(* PLC project {project_name}, OpenIXl generator OpenIXL generator v0.1 *)
(* stored: companyURL https://github.com/Bleebop/IXL_project, creationDateTime {creation_date_time}, modificationDateTime {creation_date_time} *)

TYPE TC : (NIL := -1);
END_TYPE

TYPE SWITCH : (NIL := -1);
END_TYPE

TYPE SIGNAL : (NIL := -1);
END_TYPE

TYPE TRAIN_STATE : STRUCT
  exists : BOOL;
  rear_pos : TC;
  front_pos : TC;
  orientation : DIR;
  stopped : BOOL;
END_STRUCT;
END_TYPE

TYPE DIR : (NIL := -1, DOWN := 0, UP := 1);
END_TYPE

TYPE SW_POS_t : (NIL := -1, LEFT := 1, RIGHT := 2, INTERMEDIATE := 3);
END_TYPE

TYPE ENTRY_POINT_t : STRUCT
  tc : TC;
  orientation : DIR;
END_STRUCT;
END_TYPE

TYPE EXIT_POINT_t : STRUCT
  tc : TC;
  orientation : DIR;
END_STRUCT;
END_TYPE

TYPE ROUTE : (NIL := -1);
END_TYPE

PROGRAM safety_PLC
  VAR
    route_state : ARRAY[1..const_g.nRoute] OF route_state;
    Approaching_train : ARRAY[1..const_g.nRoute] OF Approaching_train;
    switch_locked : ARRAY[1..const_g.nSwitch] OF BOOL;
    switch_required_left : ARRAY[1..const_g.nSwitch] OF BOOL;
    switch_required_right : ARRAY[1..const_g.nSwitch] OF BOOL;
  END_VAR
  VAR CONSTANT
    DELAY_DESTRUCT : ARRAY[1..const_g.nRoute] OF TIME := [];
  END_VAR
  VAR_OUTPUT
    route_open : ARRAY[1..const_g.nRoute] OF BOOL;
    route_entry_authorization : ARRAY[1..const_g.nRoute] OF BOOL;  (* The starting signal of the route can be opened to go through this route *)
    signal_open_maneuver : ARRAY[1..const_g.nSignal] OF BOOL;  (* Signal is opened for CBTC trains (downstream block occupation is ignored) *)
    switch_command_left : ARRAY[1..const_g.nSwitch] OF BOOL;
    switch_command_right : ARRAY[1..const_g.nSwitch] OF BOOL;
  END_VAR

(* FBD diagram, written out as Structured Text *)
END_PROGRAM

FUNCTION_BLOCK route_state
  VAR_INPUT
    route_formation_demand : BOOL;
    incompatible_routes_demand : BOOL;
    incompatible_routes_opened : BOOL;
    route_destruction_demand : BOOL;
    Transit_TCs_free : BOOL;
    risk_of_approaching_train : BOOL;
  END_VAR
  VAR
    SR_route : SR;
  END_VAR
  VAR_OUTPUT
    route_open : BOOL;
  END_VAR

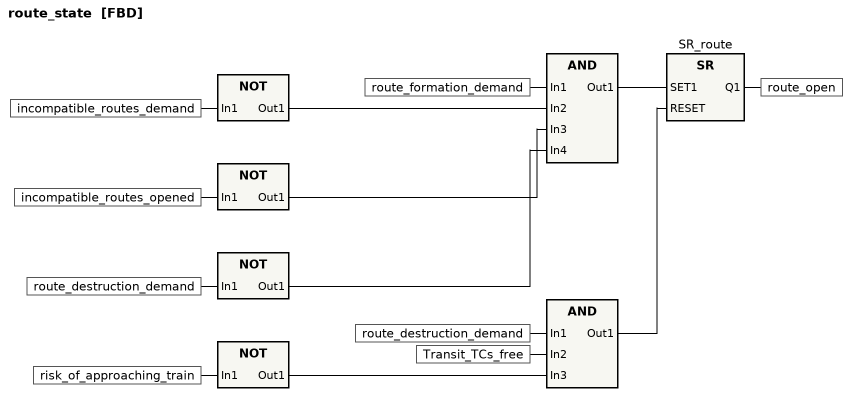
(* FBD diagram, written out as Structured Text *)
SR_route(SET1 := route_formation_demand AND NOT incompatible_routes_demand AND NOT incompatible_routes_opened AND NOT route_destruction_demand, RESET := route_destruction_demand AND Transit_TCs_free AND NOT risk_of_approaching_train);
route_open := SR_route.Q1;
END_FUNCTION_BLOCK

FUNCTION_BLOCK Approaching_train
  VAR_INPUT
    approach_area_occupied : BOOL;
    origin_signal_open : BOOL;
    DELAY_DESTRUCT : TIME;
    route_destruction_approach_ack : BOOL;
  END_VAR
  VAR_OUTPUT
    risk_of_approaching_train : BOOL;
  END_VAR
  VAR
    TON_approach_timer : TON;
    SR_approaching_train : SR;
  END_VAR

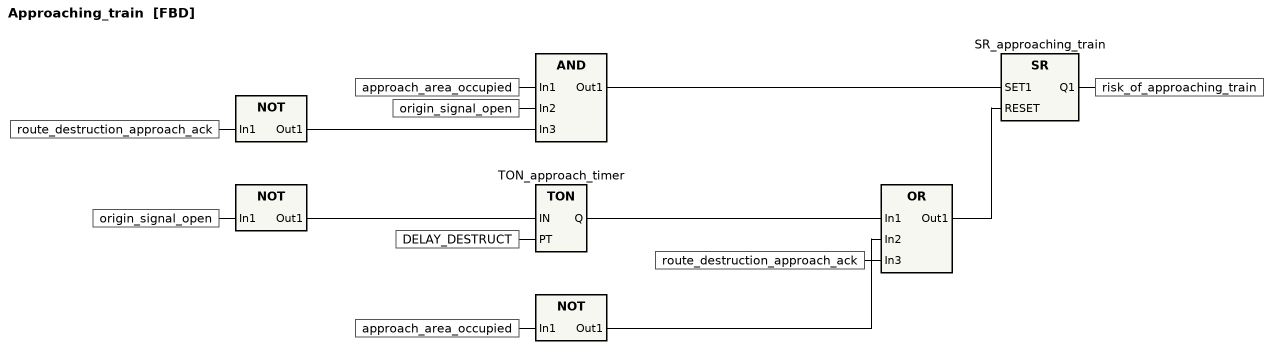
(* FBD diagram, written out as Structured Text *)
TON_approach_timer(IN := NOT origin_signal_open, PT := DELAY_DESTRUCT);
SR_approaching_train(SET1 := approach_area_occupied AND origin_signal_open AND NOT route_destruction_approach_ack, RESET := TON_approach_timer.Q OR NOT approach_area_occupied OR route_destruction_approach_ack);
risk_of_approaching_train := SR_approaching_train.Q1;
END_FUNCTION_BLOCK

CONFIGURATION Device
  RESOURCE Application ON PLC
    VAR_GLOBAL  (* var_g *)
      TC_occupied : ARRAY[1..const_g.nTC] OF BOOL;  (* /!\ safety critical /!\ *)
      switch_detected_left : ARRAY[1..const_g.nSwitch] OF BOOL;  (* /!\ safety critical /!\ *)
      switch_detected_right : ARRAY[1..const_g.nSwitch] OF BOOL;  (* /!\ safety critical /!\ *)
      switch_manual_override : ARRAY[1..const_g.nSwitch] OF BOOL;  (* Allows a switch to be moved on site /!\ safety critical /!\ *)
      close_command : ARRAY[1..const_g.nSignal] OF BOOL;  (* Force a signal to be closed *)
      ignore_TC_occupation : ARRAY[1..const_g.nTC] OF BOOL;  (* Allow to destruct a route even if this TC is occupied. /!\ safety critical /!\ *)
      ignore_approach : ARRAY[1..const_g.nRoute] OF BOOL;  (* Allow to destruct a route even if there is a risk of a train entering. /!\ safety critical /!\ *)
      route_formation_demand : ARRAY[1..const_g.nRoute] OF BOOL;
      route_destruction_demand : ARRAY[1..const_g.nRoute] OF BOOL;
    END_VAR
    VAR_GLOBAL CONSTANT  (* const_g *)
      nTC : INT := {n_tvd};  (* Track Circuits used by the IXL *)
      nRoute : INT := {n_route};  (* Routes that can be formed and destroyed *)
      nSwitch : INT := {n_switch};
      nSignal : INT := {n_signal};
    END_VAR
    TASK MainTask(INTERVAL := {plc_period}, PRIORITY := 1);
    PROGRAM safety_PLC WITH MainTask : safety_PLC;
  END_RESOURCE
END_CONFIGURATION
